(* IEC 61131-3 sources: mect_apps/TPAC1007/Local_IO_PLC, 8 files *)

(* ---- Crosstable.gvl ---- *)
VAR_GLOBAL
START_REMOTE AT %IX0.15996.0:BOOL;
START_TEST AT %IX0.16000.0:BOOL;
TST_DigIn_1 AT %IX0.16004.0:BOOL;
TST_DigIn_2 AT %IX0.16008.0:BOOL;
TST_DigIn_3 AT %IX0.16012.0:BOOL;
TST_DigIn_4 AT %IX0.16016.0:BOOL;
TST_DigIn_5 AT %IX0.16020.0:BOOL;
TST_DigIn_6 AT %IX0.16024.0:BOOL;
TST_DigIn_7 AT %IX0.16028.0:BOOL;
TST_DigIn_8 AT %IX0.16032.0:BOOL;
TST_DigIn_9 AT %IX0.16036.0:BOOL;
TST_DigIn_10 AT %IX0.16040.0:BOOL;
TST_DigIn_11 AT %IX0.16044.0:BOOL;
TST_DigIn_12 AT %IX0.16048.0:BOOL;
TST_DigIn_13 AT %IX0.16052.0:BOOL;
TST_DigIn_14 AT %IX0.16056.0:BOOL;
TST_DigIn_15 AT %IX0.16060.0:BOOL;
TST_DigIn_16 AT %IX0.16064.0:BOOL;
VAL_DigIn_1 AT %IX0.16068.0:BOOL;
VAL_DigIn_2 AT %IX0.16072.0:BOOL;
VAL_DigIn_3 AT %IX0.16076.0:BOOL;
VAL_DigIn_4 AT %IX0.16080.0:BOOL;
VAL_DigIn_5 AT %IX0.16084.0:BOOL;
VAL_DigIn_6 AT %IX0.16088.0:BOOL;
VAL_DigIn_7 AT %IX0.16092.0:BOOL;
VAL_DigIn_8 AT %IX0.16096.0:BOOL;
VAL_DigIn_9 AT %IX0.16100.0:BOOL;
VAL_DigIn_10 AT %IX0.16104.0:BOOL;
VAL_DigIn_11 AT %IX0.16108.0:BOOL;
VAL_DigIn_12 AT %IX0.16112.0:BOOL;
VAL_DigIn_13 AT %IX0.16116.0:BOOL;
VAL_DigIn_14 AT %IX0.16120.0:BOOL;
VAL_DigIn_15 AT %IX0.16124.0:BOOL;
VAL_DigIn_16 AT %IX0.16128.0:BOOL;
RES_DigIn_1 AT %QX0.16132.0:BOOL;
RES_DigIn_2 AT %QX0.16136.0:BOOL;
RES_DigIn_3 AT %QX0.16140.0:BOOL;
RES_DigIn_4 AT %QX0.16144.0:BOOL;
RES_DigIn_5 AT %QX0.16148.0:BOOL;
RES_DigIn_6 AT %QX0.16152.0:BOOL;
RES_DigIn_7 AT %QX0.16156.0:BOOL;
RES_DigIn_8 AT %QX0.16160.0:BOOL;
RES_DigIn_9 AT %QX0.16164.0:BOOL;
RES_DigIn_10 AT %QX0.16168.0:BOOL;
RES_DigIn_11 AT %QX0.16172.0:BOOL;
RES_DigIn_12 AT %QX0.16176.0:BOOL;
RES_DigIn_13 AT %QX0.16180.0:BOOL;
RES_DigIn_14 AT %QX0.16184.0:BOOL;
RES_DigIn_15 AT %QX0.16188.0:BOOL;
RES_DigIn_16 AT %QX0.16192.0:BOOL;
TST_DigOut_1 AT %IX0.16196.0:BOOL;
TST_DigOut_2 AT %IX0.16200.0:BOOL;
TST_DigOut_3 AT %IX0.16204.0:BOOL;
TST_DigOut_4 AT %IX0.16208.0:BOOL;
TST_DigOut_5 AT %IX0.16212.0:BOOL;
TST_DigOut_6 AT %IX0.16216.0:BOOL;
TST_DigOut_7 AT %IX0.16220.0:BOOL;
TST_DigOut_8 AT %IX0.16224.0:BOOL;
TST_DigOut_9 AT %IX0.16228.0:BOOL;
TST_DigOut_10 AT %IX0.16232.0:BOOL;
TST_DigOut_11 AT %IX0.16236.0:BOOL;
TST_DigOut_12 AT %IX0.16240.0:BOOL;
TST_DigOut_13 AT %IX0.16244.0:BOOL;
TST_DigOut_14 AT %IX0.16248.0:BOOL;
TST_DigOut_15 AT %IX0.16252.0:BOOL;
TST_DigOut_16 AT %IX0.16256.0:BOOL;
VAL_DigOut_1 AT %IX0.16260.0:BOOL;
VAL_DigOut_2 AT %IX0.16264.0:BOOL;
VAL_DigOut_3 AT %IX0.16268.0:BOOL;
VAL_DigOut_4 AT %IX0.16272.0:BOOL;
VAL_DigOut_5 AT %IX0.16276.0:BOOL;
VAL_DigOut_6 AT %IX0.16280.0:BOOL;
VAL_DigOut_7 AT %IX0.16284.0:BOOL;
VAL_DigOut_8 AT %IX0.16288.0:BOOL;
VAL_DigOut_9 AT %IX0.16292.0:BOOL;
VAL_DigOut_10 AT %IX0.16296.0:BOOL;
VAL_DigOut_11 AT %IX0.16300.0:BOOL;
VAL_DigOut_12 AT %IX0.16304.0:BOOL;
VAL_DigOut_13 AT %IX0.16308.0:BOOL;
VAL_DigOut_14 AT %IX0.16312.0:BOOL;
VAL_DigOut_15 AT %IX0.16316.0:BOOL;
VAL_DigOut_16 AT %IX0.16320.0:BOOL;
RES_DigOut_1 AT %QX0.16324.0:BOOL;
RES_DigOut_2 AT %QX0.16328.0:BOOL;
RES_DigOut_3 AT %QX0.16332.0:BOOL;
RES_DigOut_4 AT %QX0.16336.0:BOOL;
RES_DigOut_5 AT %QX0.16340.0:BOOL;
RES_DigOut_6 AT %QX0.16344.0:BOOL;
RES_DigOut_7 AT %QX0.16348.0:BOOL;
RES_DigOut_8 AT %QX0.16352.0:BOOL;
RES_DigOut_9 AT %QX0.16356.0:BOOL;
RES_DigOut_10 AT %QX0.16360.0:BOOL;
RES_DigOut_11 AT %QX0.16364.0:BOOL;
RES_DigOut_12 AT %QX0.16368.0:BOOL;
RES_DigOut_13 AT %QX0.16372.0:BOOL;
RES_DigOut_14 AT %QX0.16376.0:BOOL;
RES_DigOut_15 AT %QX0.16380.0:BOOL;
RES_DigOut_16 AT %QX0.16384.0:BOOL;
TST_AnIn_1 AT %IX0.16388.0:BOOL;
TST_AnIn_2 AT %IX0.16392.0:BOOL;
TST_AnIn_3 AT %IX0.16396.0:BOOL;
TST_AnIn_4 AT %IX0.16400.0:BOOL;
TST_AnIn_5 AT %IX0.16404.0:BOOL;
TST_AnIn_6 AT %IX0.16408.0:BOOL;
TST_AnIn_7 AT %IX0.16412.0:BOOL;
TST_AnIn_8 AT %IX0.16416.0:BOOL;
TST_AnIn_9 AT %IX0.16420.0:BOOL;
TST_AnIn_10 AT %IX0.16424.0:BOOL;
TST_AnIn_11 AT %IX0.16428.0:BOOL;
TST_AnIn_12 AT %IX0.16432.0:BOOL;
VAL_AnIn_1 AT %IW0.16436:INT;
VAL_AnIn_2 AT %IW0.16440:INT;
VAL_AnIn_3 AT %IW0.16444:INT;
VAL_AnIn_4 AT %IW0.16448:INT;
VAL_AnIn_5 AT %IW0.16452:INT;
VAL_AnIn_6 AT %IW0.16456:INT;
VAL_AnIn_7 AT %IW0.16460:INT;
VAL_AnIn_8 AT %IW0.16464:INT;
VAL_AnIn_9 AT %IW0.16468:INT;
VAL_AnIn_10 AT %IW0.16472:INT;
VAL_AnIn_11 AT %IW0.16476:INT;
VAL_AnIn_12 AT %IW0.16480:INT;
VAL_AnInConf_1 AT %IW0.16484:UINT;
VAL_AnInConf_2 AT %IW0.16488:UINT;
VAL_AnInConf_3 AT %IW0.16492:UINT;
VAL_AnInConf_4 AT %IW0.16496:UINT;
VAL_AnInConf_5 AT %IW0.16500:UINT;
VAL_AnInConf_6 AT %IW0.16504:UINT;
VAL_AnInConf_7 AT %IW0.16508:UINT;
VAL_AnInConf_8 AT %IW0.16512:UINT;
VAL_AnInConf_9 AT %IW0.16516:UINT;
VAL_AnInConf_10 AT %IW0.16520:UINT;
VAL_AnInConf_11 AT %IW0.16524:UINT;
VAL_AnInConf_12 AT %IW0.16528:UINT;
VAL_AnInFltr_1 AT %IW0.16532:UINT;
VAL_AnInFltr_2 AT %IW0.16536:UINT;
VAL_AnInFltr_3 AT %IW0.16540:UINT;
VAL_AnInFltr_4 AT %IW0.16544:UINT;
VAL_AnInFltr_5 AT %IW0.16548:UINT;
VAL_AnInFltr_6 AT %IW0.16552:UINT;
VAL_AnInFltr_7 AT %IW0.16556:UINT;
VAL_AnInFltr_8 AT %IW0.16560:UINT;
VAL_AnInFltr_9 AT %IW0.16564:UINT;
VAL_AnInFltr_10 AT %IW0.16568:UINT;
VAL_AnInFltr_11 AT %IW0.16572:UINT;
VAL_AnInFltr_12 AT %IW0.16576:UINT;
RES_AnIn_1 AT %QW0.16580:INT;
RES_AnIn_2 AT %QW0.16584:INT;
RES_AnIn_3 AT %QW0.16588:INT;
RES_AnIn_4 AT %QW0.16592:INT;
RES_AnIn_5 AT %QW0.16596:INT;
RES_AnIn_6 AT %QW0.16600:INT;
RES_AnIn_7 AT %QW0.16604:INT;
RES_AnIn_8 AT %QW0.16608:INT;
RES_AnIn_9 AT %QW0.16612:INT;
RES_AnIn_10 AT %QW0.16616:INT;
RES_AnIn_11 AT %QW0.16620:INT;
RES_AnIn_12 AT %QW0.16624:INT;
RES_AnInStts_1 AT %QW0.16628:INT;
RES_AnInStts_2 AT %QW0.16632:INT;
RES_AnInStts_3 AT %QW0.16636:INT;
RES_AnInStts_4 AT %QW0.16640:INT;
RES_AnInStts_5 AT %QW0.16644:INT;
RES_AnInStts_6 AT %QW0.16648:INT;
RES_AnInStts_7 AT %QW0.16652:INT;
RES_AnInStts_8 AT %QW0.16656:INT;
RES_AnInStts_9 AT %QW0.16660:INT;
RES_AnInStts_10 AT %QW0.16664:INT;
RES_AnInStts_11 AT %QW0.16668:INT;
RES_AnInStts_12 AT %QW0.16672:INT;
TST_AnOut_1 AT %IX0.16676.0:BOOL;
TST_AnOut_2 AT %IX0.16680.0:BOOL;
TST_AnOut_3 AT %IX0.16684.0:BOOL;
TST_AnOut_4 AT %IX0.16688.0:BOOL;
VAL_AnOut_1 AT %IW0.16692:INT;
VAL_AnOut_2 AT %IW0.16696:INT;
VAL_AnOut_3 AT %IW0.16700:INT;
VAL_AnOut_4 AT %IW0.16704:INT;
VAL_AnOutConf_1 AT %IW0.16708:UINT;
VAL_AnOutConf_2 AT %IW0.16712:UINT;
VAL_AnOutConf_3 AT %IW0.16716:UINT;
VAL_AnOutConf_4 AT %IW0.16720:UINT;
RES_AnOutStts_1 AT %QW0.16724:INT;
RES_AnOutStts_2 AT %QW0.16728:INT;
RES_AnOutStts_3 AT %QW0.16732:INT;
RES_AnOutStts_4 AT %QW0.16736:INT;
TST_Tamb AT %IX0.16740.0:BOOL;
TST_RPM AT %IX0.16744.0:BOOL;
TST_FWrevision AT %IX0.16748.0:BOOL;
TST_HWconfig AT %IX0.16752.0:BOOL;
VAL_Tamb AT %IW0.16756:INT;
VAL_RPM AT %IW0.16760:UINT;
VAL_FWrevision AT %IW0.16764:UINT;
VAL_HWconfig AT %IW0.16768:UINT;
RES_Tamb AT %QW0.16772:INT;
RES_RPM AT %QW0.16776:UINT;
RES_FWrevision AT %QW0.16780:UINT;
RES_HWconfig AT %QW0.16784:UINT;
TST_RTUS_WR AT %IX0.16788.0:BOOL;
TST_RTUS_RD AT %IX0.16792.0:BOOL;
TST_RTU_WR AT %IX0.16796.0:BOOL;
TST_RTU_RD AT %IX0.16800.0:BOOL;
TST_RTU3_WR AT %IX0.16804.0:BOOL;
TST_RTU3_RD AT %IX0.16808.0:BOOL;
TST_CAN_WR AT %IX0.16812.0:BOOL;
TST_CAN_RD AT %IX0.16816.0:BOOL;
VAL_RTUS_WR AT %IX0.16820.0:BOOL;
VAL_RTUS_RD AT %IX0.16824.0:BOOL;
VAL_RTU_WR AT %IX0.16828.0:BOOL;
VAL_RTU_RD AT %IX0.16832.0:BOOL;
VAL_RTU3_WR AT %IX0.16836.0:BOOL;
VAL_RTU3_RD AT %IX0.16840.0:BOOL;
VAL_CAN_WR AT %IX0.16844.0:BOOL;
VAL_CAN_RD AT %IX0.16848.0:BOOL;
RES_RTUS_WR AT %QX0.16852.0:BOOL;
RES_RTUS_RD AT %QX0.16856.0:BOOL;
RES_RTU_WR AT %QX0.16860.0:BOOL;
RES_RTU_RD AT %QX0.16864.0:BOOL;
RES_RTU3_WR AT %QX0.16868.0:BOOL;
RES_RTU3_RD AT %QX0.16872.0:BOOL;
RES_CAN_WR AT %QX0.16876.0:BOOL;
RES_CAN_RD AT %QX0.16880.0:BOOL;
STATUS_LOCAL AT %QX0.16884.0:BOOL;
STATUS_REMOTE AT %QX0.16888.0:BOOL;
STATUS_DONE AT %QX0.16892.0:BOOL;
PLC_FWrevision AT %IW0.21200:UINT;
PLC_HWconfig AT %IW0.21204:UINT;
PLC_DigDir_1 AT %QX0.21208.0:BOOL;
PLC_DigDir_2 AT %QX0.21212.0:BOOL;
PLC_DigDir_3 AT %QX0.21216.0:BOOL;
PLC_DigDir_4 AT %QX0.21220.0:BOOL;
PLC_DigDir_5 AT %QX0.21224.0:BOOL;
PLC_DigDir_6 AT %QX0.21228.0:BOOL;
PLC_DigDir_7 AT %QX0.21232.0:BOOL;
PLC_DigDir_8 AT %QX0.21236.0:BOOL;
PLC_AnInConf_1 AT %QW0.21240:UINT;
PLC_AnInConf_2 AT %QW0.21244:UINT;
PLC_AnOutConf_1 AT %QW0.21248:UINT;
PLC_DigIn_1 AT %IX0.21252.0:BOOL;
PLC_DigIn_2 AT %IX0.21256.0:BOOL;
PLC_DigIn_3 AT %IX0.21260.0:BOOL;
PLC_DigIn_4 AT %IX0.21264.0:BOOL;
PLC_DigIn_5 AT %IX0.21268.0:BOOL;
PLC_DigIn_6 AT %IX0.21272.0:BOOL;
PLC_DigIn_7 AT %IX0.21276.0:BOOL;
PLC_DigIn_8 AT %IX0.21280.0:BOOL;
PLC_DigIn_9 AT %IX0.21284.0:BOOL;
PLC_DigIn_10 AT %IX0.21288.0:BOOL;
PLC_DigIn_11 AT %IX0.21292.0:BOOL;
PLC_DigIn_12 AT %IX0.21296.0:BOOL;
PLC_AnIn_1 AT %IW0.21300:INT;
PLC_AnIn_2 AT %IW0.21304:INT;
PLC_Tamb AT %IW0.21308:INT;
PLC_Encoder AT %ID0.21312:UDINT;
PLC_DigOut_1 AT %QX0.21316.0:BOOL;
PLC_DigOut_2 AT %QX0.21320.0:BOOL;
PLC_DigOut_3 AT %QX0.21324.0:BOOL;
PLC_DigOut_4 AT %QX0.21328.0:BOOL;
PLC_DigOut_5 AT %QX0.21332.0:BOOL;
PLC_DigOut_6 AT %QX0.21336.0:BOOL;
PLC_DigOut_7 AT %QX0.21340.0:BOOL;
PLC_DigOut_8 AT %QX0.21344.0:BOOL;
PLC_AnOut_1 AT %QW0.21348:INT;
PLC_EncEnable AT %QW0.21352:UINT;
PLC_EncoderReset AT %QW0.21356:UINT;
PLC_Reserved_16 AT %QW0.21360:UINT;
PLC_Reserved_17 AT %QW0.21364:UINT;
PLC_Reserved_18 AT %QW0.21368:UINT;
PLC_Reserved_19 AT %QW0.21372:UINT;
PLC_Heartbeat AT %IW0.21376:UINT;
PLC_time AT %ID0.21560:REAL;
PLC_timeMin AT %ID0.21564:REAL;
PLC_timeMax AT %ID0.21568:REAL;
PLC_timeWin AT %QD0.21572:REAL;
END_VAR

(* ---- Resource1.gvl ---- *)
(*Global variable file*)
(*[[
]]*)
VAR_GLOBAL

END_VAR

(* ---- Alarms.st ---- *)
(*[[
]]*)
PROGRAM Alarms

#import "Resource1.gvl"
#import "Crosstable.gvl"

	;

END_PROGRAM

(* ---- Fast.st ---- *)
(*[[
]]*)
PROGRAM Fast
#import "Resource1.gvl"
#import "Crosstable.gvl"

	;

END_PROGRAM

(* ---- Initialize.st ---- *)
(*[[
]]*)
PROGRAM Initialize
#import "Resource1.gvl"
#import "Crosstable.gvl"

		(* digital i/o configuration *)
		PLC_DigDir_1 := 1; (* output *)
		PLC_DigDir_2 := 1; (* output *)
		PLC_DigDir_3 := 1; (* output *)
		PLC_DigDir_4 := 1; (* output *)
		PLC_DigDir_5 := 0; (* input *)
		PLC_DigDir_6 := 0; (* input *)
		PLC_DigDir_7 := 0; (* input *)
		PLC_DigDir_8 := 0; (* input *)

		(* analog i/o configuration *)
		PLC_AnInConf_1 := 2; (* voltage *)
		PLC_AnInConf_2 := 2; (* voltage *)
		PLC_AnOutConf_1 := 2; (* voltage *)

END_PROGRAM

(* ---- Normal.st ---- *)
(*[[
]]*)
PROGRAM Normal
#import "Resource1.gvl"
#import "Crosstable.gvl"

	PLC_AnOut_1 := ((PLC_AnIn_1 + PLC_AnIn_2) / 2) / 10;

END_PROGRAM

(* ---- Program1.st ---- *)
(*[[
]]*)
PROGRAM Program1
#import "Resource1.gvl"
#import "Crosstable.gvl"
VAR
	first : BOOL := TRUE;
	timer : TON;
	flip :BOOL := TRUE;
END_VAR;

	if first then
		(* digital i/o configuration *)
		PLC_DigDir_1 := 1; (* output *)
		PLC_DigDir_2 := 1; (* output *)
		PLC_DigDir_3 := 1; (* output *)
		PLC_DigDir_4 := 1; (* output *)
		PLC_DigDir_5 := 0; (* input *)
		PLC_DigDir_6 := 0; (* input *)
		PLC_DigDir_7 := 1; (* output *)
		PLC_DigDir_8 := 0; (* input *)

		(* analog i/o configuration *)
		PLC_AnInConf_1 := 2; (* voltage *)
		PLC_AnInConf_2 := 2; (* voltage *)
		PLC_AnOutConf_1 := 2; (* voltage *)

		first := FALSE;
	end_if;

	(* Output Action *)
	timer(IN := true, PT := T#1000ms);
	PLC_AnOut_1 := ((PLC_AnIn_1 + PLC_AnIn_2) / 2) / 10;
	if timer.Q then
		flip := not flip;
		PLC_DigOut_7 := flip;
		timer(IN := false);
	end_if;

END_PROGRAM

(* ---- Slow.st ---- *)
(*[[
]]*)
PROGRAM Slow
#import "Resource1.gvl"
#import "Crosstable.gvl"
VAR
	flip :BOOL := TRUE;
END_VAR;

		flip := not flip;
		(* Arming the Latency Test: see Task2_Alarms *)
		PLC_DigOut_1 := flip;

END_PROGRAM
